FUNCTION_BLOCK FB_Blink
VAR_INPUT
	Enable	:BOOL;
	onTime	:TIME;
	offTime	:TIME;
END_VAR
VAR_OUTPUT
	out		:BOOL;
END_VAR
VAR
	tonOff,tonOn	:TON;
END_VAR

tonOff(IN:=NOT tonOn.Q AND Enable , PT:=offTime , Q=>out );
tonOn(IN:=tonOff.Q , PT:=onTime );

END_FUNCTION_BLOCK

(* stored: Version 1.1.0.1, ProductVersion 3.1.4024.12
   POU FB_Blink: Id {a477d05d-d6a8-45eb-911d-87c7c1ce658b}, SpecialFunc None *)
